// TIA Portal V16 export
// export: Created 2025-10-06T17:54:28.6507115Z, ExportSetting WithDefaults, DisplayName Totally Integrated Automation Portal, DisplayVersion V16, DisplayName TIA Portal Version Control Interface, DisplayVersion V16, DisplayName TIA Portal Openness, DisplayVersion V16, DisplayName STEP 7 Professional, DisplayVersion V16, DisplayName STEP 7 Safety, DisplayVersion V16, DisplayName WinCC Advanced, DisplayVersion V16
FUNCTION_BLOCK "TestingAndOld"   // FB24, LAD
VERSION : 0.1
// stored: AutoNumber true, IsIECCheckEnabled false, UDAEnableTagReadback false
   VAR_TEMP
      NotUsed : Bool;
      SAFE_OK_Signal : Bool;
      ScPos : Real;
      ActEncPos : Real;
      DB : Real;
   END_VAR
BEGIN

REGION Network 2: Encoder Feedback Connection FB
   // Getting the feedback from the encoder device
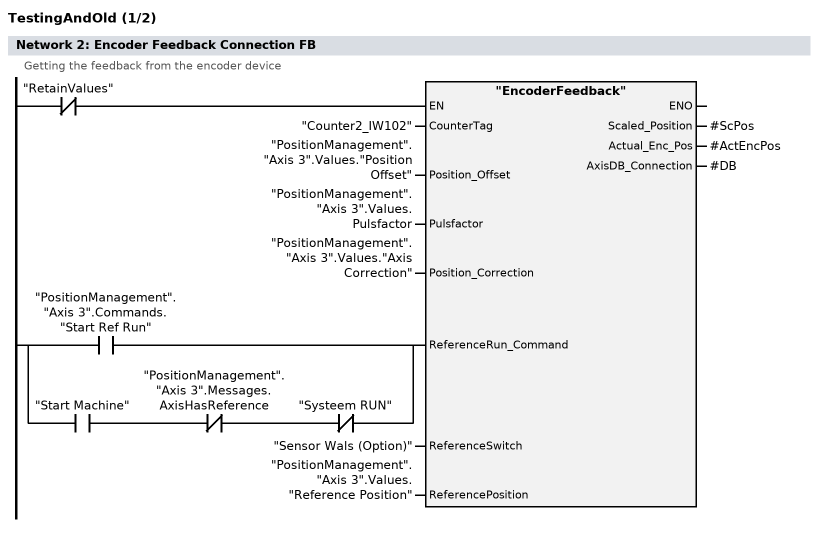
   RUNG wire#powerrail
      I_Contact( "RetainValues" )
      "EncoderFeedback"(ReferenceRun_Command := wire#w1, CounterTag := "Counter2_IW102", Position_Offset := "PositionManagement"."Axis 3".Values."Position Offset", Pulsfactor := "PositionManagement"."Axis 3".Values.Pulsfactor, Position_Correction := "PositionManagement"."Axis 3".Values."Axis Correction", ReferenceSwitch := "Sensor Wals (Option)", ReferencePosition := "PositionManagement"."Axis 3".Values."Reference Position", Scaled_Position => #ScPos, Actual_Enc_Pos => #ActEncPos, AxisDB_Connection => #DB)
   END_RUNG
   RUNG wire#powerrail
      Contact( "PositionManagement"."Axis 3".Commands."Start Ref Run" )
   END_RUNG wire#w1
   RUNG wire#powerrail
      Contact( "Start Machine" )
      I_Contact( "PositionManagement"."Axis 3".Messages.AxisHasReference )
      I_Contact( "Systeem RUN" )
   END_RUNG wire#w1
   // the same network as SCL:
   IF NOT "RetainValues" THEN
       "EncoderFeedback"(CounterTag := "Counter2_IW102",
                         Position_Offset := "PositionManagement"."Axis 3".Values."Position Offset",
                         Pulsfactor := "PositionManagement"."Axis 3".Values.Pulsfactor,
                         Position_Correction := "PositionManagement"."Axis 3".Values."Axis Correction",
                         ReferenceRun_Command := "PositionManagement"."Axis 3".Commands."Start Ref Run" OR ("Start Machine" AND NOT "PositionManagement"."Axis 3".Messages.AxisHasReference AND NOT "Systeem RUN"),
                         ReferenceSwitch := "Sensor Wals (Option)",
                         ReferencePosition := "PositionManagement"."Axis 3".Values."Reference Position",
                         Scaled_Position => #ScPos,
                         Actual_Enc_Pos => #ActEncPos,
                         AxisDB_Connection => #DB);
   END_IF;
END_REGION

REGION Network 3: Drive Manager Axis 3
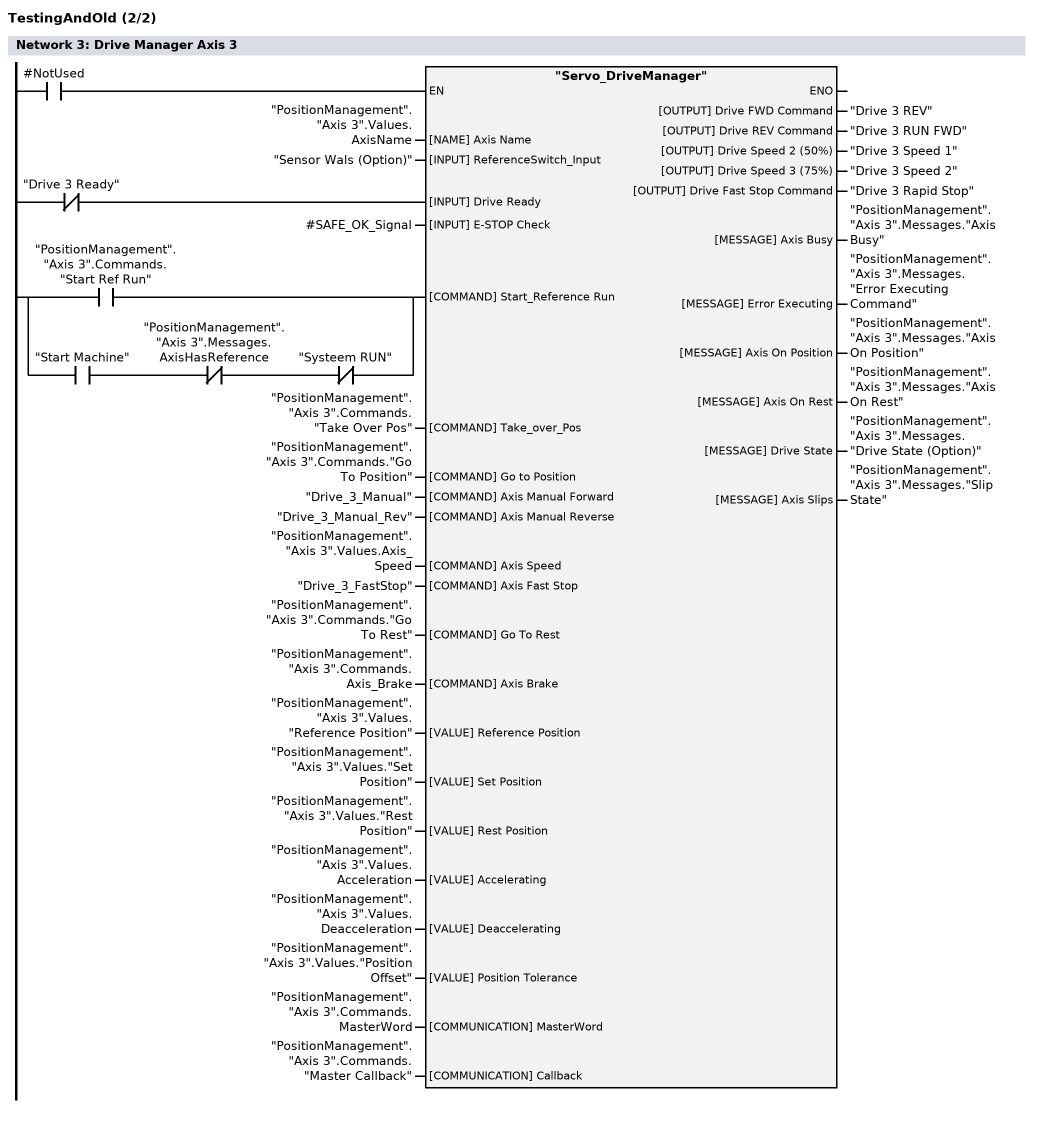
   RUNG wire#powerrail
      Contact( #NotUsed )
      "Servo_DriveManager"("[INPUT] Drive Ready" := wire#w1, "[COMMAND] Start_Reference Run" := wire#w2, "[NAME] Axis Name" := "PositionManagement"."Axis 3".Values.AxisName, "[INPUT] ReferenceSwitch_Input" := "Sensor Wals (Option)", "[INPUT] E-STOP Check" := #SAFE_OK_Signal, "[COMMAND] Take_over_Pos" := "PositionManagement"."Axis 3".Commands."Take Over Pos", "[COMMAND] Go to Position" := "PositionManagement"."Axis 3".Commands."Go To Position", "[COMMAND] Axis Manual Forward" := "Drive_3_Manual", "[COMMAND] Axis Manual Reverse" := "Drive_3_Manual_Rev", "[COMMAND] Axis Speed" := "PositionManagement"."Axis 3".Values.Axis_Speed, "[COMMAND] Axis Fast Stop" := "Drive_3_FastStop", "[COMMAND] Go To Rest" := "PositionManagement"."Axis 3".Commands."Go To Rest", "[COMMAND] Axis Brake" := "PositionManagement"."Axis 3".Commands.Axis_Brake, "[VALUE] Reference Position" := "PositionManagement"."Axis 3".Values."Reference Position", "[VALUE] Set Position" := "PositionManagement"."Axis 3".Values."Set Position", "[VALUE] Rest Position" := "PositionManagement"."Axis 3".Values."Rest Position", "[VALUE] Accelerating" := "PositionManagement"."Axis 3".Values.Acceleration, "[VALUE] Deaccelerating" := "PositionManagement"."Axis 3".Values.Deacceleration, "[VALUE] Position Tolerance" := "PositionManagement"."Axis 3".Values."Position Offset", "[COMMUNICATION] MasterWord" := "PositionManagement"."Axis 3".Commands.MasterWord, "[COMMUNICATION] Callback" := "PositionManagement"."Axis 3".Commands."Master Callback", "[OUTPUT] Drive FWD Command" => "Drive 3 REV", "[OUTPUT] Drive REV Command" => "Drive 3 RUN FWD", "[OUTPUT] Drive Speed 2 (50%)" => "Drive 3 Speed 1", "[OUTPUT] Drive Speed 3 (75%)" => "Drive 3 Speed 2", "[OUTPUT] Drive Fast Stop Command" => "Drive 3 Rapid Stop", "[MESSAGE] Axis Busy" => "PositionManagement"."Axis 3".Messages."Axis Busy", "[MESSAGE] Error Executing" => "PositionManagement"."Axis 3".Messages."Error Executing Command", "[MESSAGE] Axis On Position" => "PositionManagement"."Axis 3".Messages."Axis On Position", "[MESSAGE] Axis On Rest" => "PositionManagement"."Axis 3".Messages."Axis On Rest", "[MESSAGE] Drive State" => "PositionManagement"."Axis 3".Messages."Drive State (Option)", "[MESSAGE] Axis Slips" => "PositionManagement"."Axis 3".Messages."Slip State")
   END_RUNG
   RUNG wire#powerrail
      I_Contact( "Drive 3 Ready" )
   END_RUNG wire#w1
   RUNG wire#powerrail
      Contact( "PositionManagement"."Axis 3".Commands."Start Ref Run" )
   END_RUNG wire#w2
   RUNG wire#powerrail
      Contact( "Start Machine" )
      I_Contact( "PositionManagement"."Axis 3".Messages.AxisHasReference )
      I_Contact( "Systeem RUN" )
   END_RUNG wire#w2
   // the same network as SCL:
   IF #NotUsed THEN
       "Servo_DriveManager"("[NAME] Axis Name" := "PositionManagement"."Axis 3".Values.AxisName,
                            "[INPUT] ReferenceSwitch_Input" := "Sensor Wals (Option)",
                            "[INPUT] Drive Ready" := NOT "Drive 3 Ready",
                            "[INPUT] E-STOP Check" := #SAFE_OK_Signal,
                            "[COMMAND] Start_Reference Run" := "PositionManagement"."Axis 3".Commands."Start Ref Run" OR ("Start Machine" AND NOT "PositionManagement"."Axis 3".Messages.AxisHasReference AND NOT "Systeem RUN"),
                            "[COMMAND] Take_over_Pos" := "PositionManagement"."Axis 3".Commands."Take Over Pos",
                            "[COMMAND] Go to Position" := "PositionManagement"."Axis 3".Commands."Go To Position",
                            "[COMMAND] Axis Manual Forward" := "Drive_3_Manual",
                            "[COMMAND] Axis Manual Reverse" := "Drive_3_Manual_Rev",
                            "[COMMAND] Axis Speed" := "PositionManagement"."Axis 3".Values.Axis_Speed,
                            "[COMMAND] Axis Fast Stop" := "Drive_3_FastStop",
                            "[COMMAND] Go To Rest" := "PositionManagement"."Axis 3".Commands."Go To Rest",
                            "[COMMAND] Axis Brake" := "PositionManagement"."Axis 3".Commands.Axis_Brake,
                            "[VALUE] Reference Position" := "PositionManagement"."Axis 3".Values."Reference Position",
                            "[VALUE] Set Position" := "PositionManagement"."Axis 3".Values."Set Position",
                            "[VALUE] Rest Position" := "PositionManagement"."Axis 3".Values."Rest Position",
                            "[VALUE] Accelerating" := "PositionManagement"."Axis 3".Values.Acceleration,
                            "[VALUE] Deaccelerating" := "PositionManagement"."Axis 3".Values.Deacceleration,
                            "[VALUE] Position Tolerance" := "PositionManagement"."Axis 3".Values."Position Offset",
                            "[COMMUNICATION] MasterWord" := "PositionManagement"."Axis 3".Commands.MasterWord,
                            "[COMMUNICATION] Callback" := "PositionManagement"."Axis 3".Commands."Master Callback",
                            "[OUTPUT] Drive FWD Command" => "Drive 3 REV",
                            "[OUTPUT] Drive REV Command" => "Drive 3 RUN FWD",
                            "[OUTPUT] Drive Speed 2 (50%)" => "Drive 3 Speed 1",
                            "[OUTPUT] Drive Speed 3 (75%)" => "Drive 3 Speed 2",
                            "[OUTPUT] Drive Fast Stop Command" => "Drive 3 Rapid Stop",
                            "[MESSAGE] Axis Busy" => "PositionManagement"."Axis 3".Messages."Axis Busy",
                            "[MESSAGE] Error Executing" => "PositionManagement"."Axis 3".Messages."Error Executing Command",
                            "[MESSAGE] Axis On Position" => "PositionManagement"."Axis 3".Messages."Axis On Position",
                            "[MESSAGE] Axis On Rest" => "PositionManagement"."Axis 3".Messages."Axis On Rest",
                            "[MESSAGE] Drive State" => "PositionManagement"."Axis 3".Messages."Drive State (Option)",
                            "[MESSAGE] Axis Slips" => "PositionManagement"."Axis 3".Messages."Slip State");
   END_IF;
END_REGION
END_FUNCTION_BLOCK
